{attribute addProperty BoxType "EK1100-0000-0018"}
{attribute addProperty Id "Beckhoff_EK13xxEK1122Beckhoff_EK13xxEK1122_7883D180506.25A_0003_EK1322_0000_0017EK1322_0EEAC8F2344.25A_0002_EK1310_0000_0017EK1310_0EEAC8F2344.25"}
{attribute addProperty CRC "4153393400"}
{attribute addProperty SizeInBites "118"}
{attribute addProperty SizeInBytes "14.75"}
TYPE Beckhoff_EK13xx_F78FC0F8 EXTENDS EK1100_179A0949 :
STRUCT
	{attribute addProperty Name "Beckhoff_EK13xxEK1122"}
	Beckhoff_EK13xxEK1122 : Beckhoff_EK13xxEK1122_7883D180;
	{attribute addProperty Name "A_0003_EK1322_0000_0017"}
	A_0003_EK1322_0000_0017 : EK1322_0EEAC8F2;
	{attribute addProperty Name "A_0002_EK1310_0000_0017"}
	A_0002_EK1310_0000_0017 : EK1310_0EEAC8F2;
END_STRUCT
END_TYPE

(* stored: Version 1.2.0.0, ProductVersion 3.1.4024.9
   DUT Beckhoff_EK13xx_F78FC0F8: Id {4baba9a7-7f71-40d8-8f61-37d5d77ec19f} *)
